Universal Robots URScript: 00C_03_Che_ZhuaXian.script

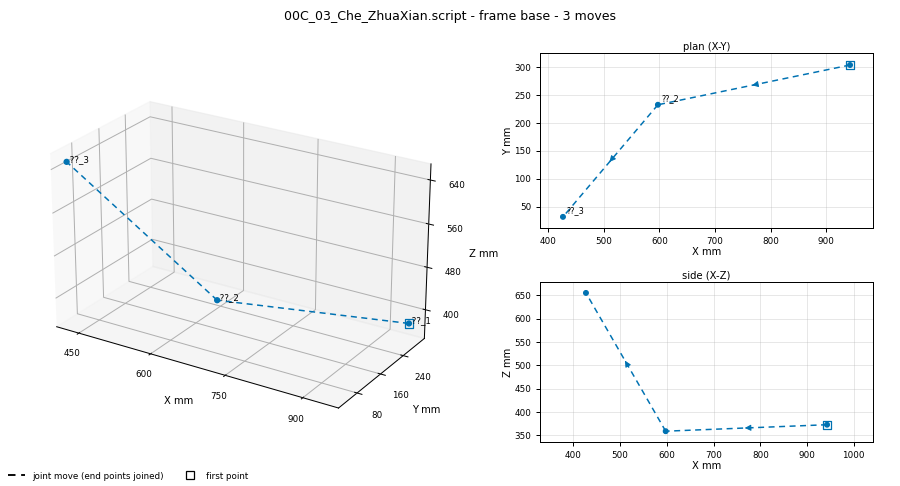
[picture p0: tool path of 00C_03_Che_ZhuaXian.script in frame base, 3 of 3 moves have a stored position in this frame; points joined in program order, loops and branches not executed]
def P00C_03_Che_ZhuaXian():
  set_standard_analog_input_domain(0, 1)
  set_standard_analog_input_domain(1, 1)
  set_tool_analog_input_domain(0, 1)
  set_tool_analog_input_domain(1, 1)
  set_analog_outputdomain(0, 0)
  set_analog_outputdomain(1, 0)
  set_tool_voltage(0)
  set_input_actions_to_default()
  set_tcp(p[-0.06448999999999999,0.0207,0.28314999999999996,0.0,0.0,1.5902])
  set_payload(8.0)
  set_safety_mode_transition_hardness(1)
  set_gravity([0.0, 0.0, 9.82])
  $ 1 "机器人程序"
  $ 2 "MoveJ"
  $ 3 "路点_1"
  set_tcp(p[-8.5E-4,0.01448,0.31003,0.0,0.0,-0.3645])
  movej(get_inverse_kin(p[.942816568158, .304387250600, .372939185917, -1.314485019015, .989248340700, -1.148649693386], qnear=[0.6537608504295349, -1.6546605269061487, -1.9450343290912073, -2.6294830481158655, -1.107157055531637, -2.8940003553973597]), a=0.6981317007977318, v=0.5235987755982988)
  $ 4 "路点_2"
  set_tcp(p[-8.5E-4,0.01448,0.31003,0.0,0.0,-0.3645])
  movej(get_inverse_kin(p[.597413541700, .232935770836, .359059025242, -1.314473794476, .989259605270, -1.148622023083], qnear=[1.319711446762085, -0.9241340796100062, -2.476755205784933, -2.774465862904684, -0.4424985090838831, -2.9616325537311]), a=0.6981317007977318, v=0.5235987755982988)
  $ 5 "路点_3"
  set_tcp(p[-8.5E-4,0.01448,0.31003,0.0,0.0,-0.3645])
  movej(get_inverse_kin(p[.426725271139, .031409999162, .655031196421, -.007988765036, .061439267686, -1.298933381599], qnear=[0.5013005137443542, -1.4665511290179651, -2.67100698152651, -0.603699032460348, -1.5243762175189417, -3.0075951258288782]), a=0.6981317007977318, v=0.5235987755982988)
end
